// TwinCAT 3 PLC project TC3_CNC
// ProgramVersion: 3.1.4023.0
// libraries:
//   Tc2_Standard, * (Beckhoff Automation GmbH)
//   Tc2_System, * (Beckhoff Automation GmbH)
//   Tc3_Module, * (Beckhoff Automation GmbH)
// project tree:
//   / PlcTask.TcTTO
//   POUs/ MAIN.TcPOU, MotionControl.TcPOU
// real-time tasks:
//   TASK PlcTask: cycle T#10ms, priority 20, ADS port 350

CONFIGURATION TC3_CNC
    RESOURCE PLC ON TwinCAT3
        TASK PlcTask(INTERVAL := T#10ms, PRIORITY := 20);
        PROGRAM MAIN WITH PlcTask : MAIN;
    END_RESOURCE
END_CONFIGURATION

// ---- POUs/MAIN.TcPOU
PROGRAM MAIN
VAR
	bInit			: 	BOOL	:=FALSE;
	bStatus			:	BOOL;
	PosControl		:	MotionControl;
	
END_VAR

IF NOT bInit THEN
	

	bInit	:=TRUE;
END_IF

END_PROGRAM

// ---- POUs/MotionControl.TcPOU
FUNCTION_BLOCK MotionControl
VAR_INPUT
END_VAR
VAR_OUTPUT
END_VAR
VAR
	cncChannnelHandler	:TC_CNC;
	refAxis		: AXIS_REF;
END_VAR

ACTION AxisControl:

END_ACTION

METHOD GetPosition : DWORD
VAR_INPUT
END_VAR
END_METHOD

METHOD setAxis : BOOL
VAR_INPUT
	refToAxis		:AXIS_REF;
END_VAR
END_METHOD

METHOD SetParams : BOOL
VAR_INPUT
END_VAR
END_METHOD

METHOD SetPosition : BOOL
VAR_INPUT
END_VAR
END_METHOD

END_FUNCTION_BLOCK
